(* CODESYS project OOP example Pointers as Arguments.project

Project tree, tasks and I/O mapping:
  Device : CODESYS Control for Raspberry Pi SL, 3S - Smart Software Solutions GmbH, version 3.5.12.30
    application Application
      libraries: Standard, * (System); VisuDialogs, * (System); SysFile, 3.5.9.0 (System); AlarmManager, 3.5.12.0 (Intern)
      task MainTask (cyclic, interval 500 ms, priority 1, watchdog 1000 ms x 1) calls Pointers_as_Argument
      program Pointers_as_Argument [ST]
    SoftMotion General Axis Pool
    I²C
    SPI
    GPIOs_A_B : GPIOs B+/Pi2, 3S - Smart Software Solutions GmbH, version 3.5.11.0
        unmapped channels: digital inputs (GPIO0..GPIO31), digital outputs (GPIO0..GPIO31)
    Onewire
    Camera device
      <Empty>
  libraries: VisuSymbols, 3.5.10.0 (System)
  Pointers as Argument/
    Handler/
      interface ITF_AlarmHandler: RegisterAlarm, ResetAllAlarms
      function block FB_AlarmHandler [ST]: RegisterAlarm, ResetAllAlarms, Registered
    Source/
      function block FB_FinalEngine [ST]: ResetAlarm, RaiseAlarm, fb_Init, Alarms
      interface ITF_AlarmSource: ResetAlarm, Alarms
      interface ITF_RaiseAlarm: RaiseAlarm
    Engines/
      function block FB_Engine [ST]: Start, Stop, MaxVelocity, Temperature, Velocity
      function block FB_NewEngine [ST]: Gear, Start
*)

// Device/Application/Pointers_as_Argument
PROGRAM Pointers_as_Argument
VAR
	AlarmHandler : FB_AlarmHandler();					// The alarmhandler, which monitors all Engine alarms
	FinalEngine1 : FB_FinalEngine( ADR(AlarmHandler) );	// Each engine registers itself at the alarmhandler (see method register alarm)
	FinalEngine2 : FB_FinalEngine( ADR(AlarmHandler) );	
	
	ResetAlms 	: BOOL := FALSE;

	AmmountRegistered : INT;
	Alm1 			: BOOL := FALSE;
	Alm2 			: BOOL := FALSE;

END_VAR

IF Alm1 THEN
	FinalEngine1.RaiseAlarm();
	Alm1 := FALSE;
END_IF

IF Alm2 THEN
	FinalEngine2.RaiseAlarm();
	Alm2 := FALSE;
END_IF

AmmountRegistered := AlarmHandler.Registered;	// every registry equals an alarm

IF ResetAlms THEN
	AlarmHandler.ResetAllAlarms();
	ResetAlms := FALSE;
END_IF

END_PROGRAM

// Pointers as Argument/Handler/FB_AlarmHandler
FUNCTION_BLOCK FB_AlarmHandler IMPLEMENTS ITF_AlarmHandler
VAR
	_aritfDeviceList : ARRAY [0..99] OF ITF_AlarmSource;
	_iDeviceAmmount : INT := 0;
END_VAR

METHOD RegisterAlarm
VAR_INPUT
	deviceWithAlarm : ITF_AlarmSource;
END_VAR
VAR
	iLoopIndex : INT;
END_VAR
FOR iLoopIndex := 0 TO THIS^._iDeviceAmmount - 1 DO
	IF _aritfDeviceList[ iLoopIndex ] = DeviceWithAlarm THEN
		RETURN;		//  Double entry => exit
	END_IF
END_FOR

// if we did not exit, it's not a double entry..
THIS^._aritfDeviceList[ THIS^._iDeviceAmmount ] := DeviceWithAlarm;
THIS^._iDeviceAmmount := THIS^._iDeviceAmmount + 1;
END_METHOD

METHOD ResetAllAlarms
VAR
	iLoopIndex    : INT := 0;
END_VAR
//Resets all the alarms on each motor
FOR iLoopIndex := 0 TO THIS^._iDeviceAmmount - 1 DO
	IF _aritfDeviceList[ iLoopIndex ].Alarms <> 0 THEN
		_aritfDeviceList[ iLoopIndex ].ResetAlarm();	// pointer to all subscripted fb's Reset Methods
	END_IF
END_FOR
THIS^._iDeviceAmmount := 0;
END_METHOD

// function block gekoppelde property (niet via een interface)
PROPERTY Registered : INT
GET
Registered := _iDeviceAmmount;
END_GET
END_PROPERTY

END_FUNCTION_BLOCK

// Pointers as Argument/Handler/ITF_AlarmHandler
INTERFACE ITF_AlarmHandler

METHOD RegisterAlarm
VAR_INPUT
	deviceWithAlarm:   ITF_AlarmSource;
END_VAR
END_METHOD

METHOD ResetAllAlarms
VAR_INPUT
END_VAR
END_METHOD

END_INTERFACE

// Pointers as Argument/Source/ITF_AlarmSource
INTERFACE ITF_AlarmSource

METHOD ResetAlarm
VAR_INPUT
END_VAR
END_METHOD

//return the alarm ammount
PROPERTY Alarms : INT
GET
END_GET
END_PROPERTY

END_INTERFACE

// Pointers as Argument/Source/FB_FinalEngine
FUNCTION_BLOCK FINAL FB_FinalEngine EXTENDS FB_NewEngine IMPLEMENTS ITF_AlarmSource, ITF_RaiseAlarm
VAR
  	pAlarmHandler: POINTER TO FB_AlarmHandler;
	iAlarm : INT := 0;	// <>0 = alarm, ideally each implemented seperate alarm raises the alarmcounter via method RaiseAlarm
END_VAR

SUPER^();

METHOD ResetAlarm
//reset the alarm (lower semaphore)
iAlarm := iAlarm - 1;
END_METHOD

//Alarm!
METHOD RaiseAlarm
iAlarm := iAlarm + 1;									// uh ohh! raise the counter, which works like a semaphore
THIS^.pAlarmHandler^.RegisterAlarm( THIS^ );	//register myself at handler, because we got troubles
END_METHOD

METHOD fb_Init : BOOL
VAR_INPUT
	bInitRetains : BOOL; // TRUE: the retain variables are initialized (reset warm / reset cold)
	bInCopyCode : BOOL;  // TRUE the instance will be copied to the copy-code afterward (online change)
	AlarmHandler: POINTER TO FB_AlarmHandler;		
END_VAR
THIS^.pAlarmHandler := AlarmHandler;		// store the handler address
END_METHOD

//return the alarm ammount
PROPERTY Alarms : INT
GET
Alarms := THIS^.iAlarm;
END_GET
END_PROPERTY

END_FUNCTION_BLOCK

// Pointers as Argument/Engines/FB_NewEngine
FUNCTION_BLOCK FB_NewEngine EXTENDS FB_Engine

// HAS GOT 2 NEW Features;
// 1) START has been redefined and 
// 2) A new Gear accessor has been added
//
// these methods are fixed to the class
SUPER^();

// new property to get / set the gear after start
PROPERTY Gear : int
SET
THIS^._iGear := Gear;
END_SET
GET
Gear := THIS^._iGear;
END_GET
END_PROPERTY

METHOD Start : BOOL;
VAR_INPUT
   rVelocity : REAL;
   iGear     : INT;
END_VAR
// Overwriting an existing method (OVERRIDE)

// new: setting gear via property Gear setter
SUPER^.Start(iGear, TO_INT(rVelocity)); // calls Start() of FB_Engine, see below for explanation
Gear := iGear;


// SUPER^. POINTER
//In the above example, we created a new Start() METHOD in FB_NewEngine 
//and copied the existing code from FB_Engine into the new method. 
//This is not always possible, and it also runs counter to the principle of reuse!
//
//Consequently, every function block which is derived from another function block has access to a pointer called SUPER. 
//This can be used to access elements (methods, properties, local variables, etc.) from the parent function block.
//
//
//SUPER^.Start(nGear, fVelocity); // calls Start() of FB_Engine
//Gear := nGear;
//
//Instead of copying code from the parent function block to the new method, 
//the SUPER pointer can be used to call the method from the FB_Engine function block. 
//This does away with the need to copy the code. 
//So, SUPER calls the Father of a method
END_METHOD

END_FUNCTION_BLOCK

// Pointers as Argument/Engines/FB_Engine
// Class FB_Engine
FUNCTION_BLOCK FB_Engine
VAR
   _xStarted : BOOL;
   _rVelocity : REAL;
   _rMaxVelocity : REAL;
   _iGear : INT;
   _rTemperature : REAL;
END_VAR

//The THIS pointer is available to all function blocks and points to the current function block instance. 
//It is required whenever a method contains a local variable which obscures a variable in the function block.
//
//An assignment statement within the method sets the value of the local variable. 
//If we want the method to set the value of the local variable in the function block, we need to use the THIS pointer to access it.
METHOD Start : Bool;
VAR_INPUT
   rVelocity : REAL;
   iGear     : INT;
END_VAR
THIS^._xStarted  := TRUE;
Start            := TRUE;
THIS^._iGear     := iGear;
THIS^._rVelocity := MIN( ABS(THIS^._rMaxVelocity), rVelocity );

CASE TO_INT( THIS^._rVelocity ) OF // implicit typecasting(TO_INT), use REAL_TO_INT for explicit typecasting
   0..100 :
      THIS^._rTemperature := 50;
   101..1000:
      THIS^._rTemperature := 90;
   1001..10000:
      THIS^._rTemperature := 100;
   10001..32767:
      THIS^._rTemperature := 150;
END_CASE
END_METHOD

METHOD Stop : BOOL
VAR_INPUT
END_VAR
THIS^._xStarted := FALSE;
Stop            := TRUE;
END_METHOD

PROPERTY MaxVelocity : REAL
SET
THIS^._rMaxVelocity := MaxVelocity;
END_SET
GET
MaxVelocity := THIS^._rMaxVelocity;
END_GET
END_PROPERTY

PROPERTY Temperature : REAL
GET
Temperature := THIS^._rTemperature;
END_GET
END_PROPERTY

PROPERTY Velocity : real
GET
Velocity := THIS^._rVelocity;
END_GET
END_PROPERTY

END_FUNCTION_BLOCK

// Pointers as Argument/Source/ITF_RaiseAlarm
INTERFACE ITF_RaiseAlarm

METHOD RaiseAlarm
END_METHOD

END_INTERFACE
